Fanuc KAREL source: kt00899.KL

PROGRAM KT00899
%STACKSIZE=65535
%PRIORITY=65535
%NOLOCKGROUP
VAR
P1 : XYZWPR
P2 : XYZWPR
OUT : BOOLEAN
BEGIN
P1.X=1.0
P2.Y=2.0
P1.X=1.0
P2.Y=2.0
-- UNRESOLVED_PC line 12 opcodes [27 27 49 7E AD 27 9D 76 23] marker_code=80
END KT00899
